INTERFACE I_PackML_CompletingCommands

METHOD PUBLIC Abort
VAR_INPUT
END_VAR
END_METHOD

METHOD StateComplete
VAR_INPUT
END_VAR
END_METHOD

METHOD PUBLIC Stop
VAR_INPUT
END_VAR
END_METHOD

END_INTERFACE

(* stored: Version 1.1.0.1, ProductVersion 3.1.4024.12
   Itf I_PackML_CompletingCommands: Id {81f78d50-be70-0fcb-055f-f4ffcddca7b0}
   Method Abort: Id {f61706d9-5300-0d36-320f-75883bc3afd4}
   Method StateComplete: Id {154012f7-60dc-0bf8-1d8e-d74aafba0598}
   Method Stop: Id {dcc0e15d-c0e0-0a77-1986-dc07431ee026} *)
